TEXTLIST txtMotorTypes
  0 = 'Contactor'
  1 = 'FI'
   = ''
END_TEXTLIST

(* stored: Version 1.1.0.1, ProductVersion 3.1.4019.2
   TextList txtMotorTypes: Id {1243fcf6-6fa6-401c-a2e5-5fa728bb37cc} *)
